FUNCTION_BLOCK FB_StatesTest
VAR_INPUT
	xboVectorTargetReached : BOOL;
	xinSatus : INT;
END_VAR
VAR_OUTPUT
	yinControl : RobotControl;
	ysTargetPosition : sPosition;
	yinTargetMap : INT;
END_VAR
VAR
	sStates : sStatesForTest;
	tonDelayWait : TON;
	tonDelayTargetReach : TON;
END_VAR
VAR CONSTANT
	//Robby 3
	creTarget1X : REAL := 628.1;
	creTarget1Y : REAL := 2668.6;
	creTarget1Phi : REAL := 0.4;
	creTarget2X : REAL := 1067.3;
	creTarget2Y : REAL := 2672.3;
	creTarget2Phi : REAL := -179.6;
	
END_VAR

CASE sStates OF
	
	sStatesForTest.Target1Vektor : 
	Gripper.closeGripperCommand := FALSE;
		yinTargetMap := 1;
		IF xboVectorTargetReached THEN 
			sStates := sStatesForTest.CoordinatesInFrontOfTarget1;
		END_IF;
		
	sStatesForTest.CoordinatesInFrontOfTarget1 :
		ysTargetPosition.reX := creTarget1X - 100;
		ysTargetPosition.reY := creTarget1Y;
		ysTargetPosition.reWinkel := creTarget1Phi;
		IF xinSatus = 3 THEN 
			sStates := sStatesForTest.Wait1;
		END_IF;
		
	sStatesForTest.Wait1 : 
	
	

		ysTargetPosition.reX := creTarget1X;
		IF 	xinSatus = 1 AND tonDelayWait.Q THEN 
			sStates := sStatesForTest.Target1;
		END_IF
		
	sStatesForTest.Target1 :
		
		IF xinSatus = 3 THEN 
			sStates := sStatesForTest.Wait2;
		END_IF;
		
	sStatesForTest.Wait2 : 
		Gripper.closeGripperCommand := TRUE;
		ysTargetPosition.reX := creTarget1X - 100;
		IF 	xinSatus = 1 AND tonDelayWait.Q THEN 
			sStates := sStatesForTest.AfterTarget1;
		END_IF
		
	sStatesForTest.AfterTarget1 :
		
		IF xinSatus = 3 THEN 
			sStates := sStatesForTest.Target2Vector;
		END_IF;
		
	sStatesForTest.Target2Vector :
	
		yinTargetMap := 2;
		IF xboVectorTargetReached THEN 
			sStates := sStatesForTest.CoordinatesInFrontOfTarget2;
		END_IF;
		
	sStatesForTest.CoordinatesInFrontOfTarget2 :
		ysTargetPosition.reX := creTarget2X + 100;
		ysTargetPosition.reY := creTarget2Y;
		ysTargetPosition.reWinkel := creTarget2Phi;
		IF xinSatus = 3 THEN 
			sStates := sStatesForTest.Wait3;
		END_IF;
		
		sStatesForTest.Wait3 : 
		ysTargetPosition.reX := creTarget2X;
		IF 	xinSatus = 1 AND tonDelayWait.Q THEN 
			sStates := sStatesForTest.Target2;
		END_IF	
		
	sStatesForTest.Target2 :
	
		
		IF xinSatus = 3 THEN 
			sStates := sStatesForTest.Wait4;
		END_IF;
		
		
		sStatesForTest.Wait4 : 
		Gripper.closeGripperCommand := FALSE;
		ysTargetPosition.reX := creTarget2X + 100;
		IF 	xinSatus = 1 AND tonDelayWait.Q THEN 
			sStates := sStatesForTest.AfterTarget2;
		END_IF	
		
	sStatesForTest.AfterTarget2 :
	
		IF xinSatus = 3 THEN 
			sStates := sStatesForTest.ParkingVector;
		END_IF;
		
	sStatesForTest.ParkingVector :
	
		yinTargetMap := 7;
		IF xboVectorTargetReached THEN 
			sStates := sStatesForTest.Finished;
		END_IF;
		
	sStatesForTest.Finished : ;
	
END_CASE

tonDelayWait(IN := (sStatesForTest.Wait1 = sStates) OR (sStatesForTest.Wait2 = sStates) OR (sStatesForTest.Wait3 = sStates) OR (sStatesForTest.Wait4 = sStates), PT := T#0.1S);

IF (sStatesForTest.Target1Vektor = sStates) OR (sStatesForTest.Target2Vector = sStates) OR (sStatesForTest.ParkingVector = sStates) THEN
	yinControl := 3;
END_IF

IF (sStatesForTest.CoordinatesInFrontOfTarget1 = sStates) OR (sStatesForTest.Target1 = sStates) OR (sStatesForTest.AfterTarget1 = sStates)
 OR (sStatesForTest.CoordinatesInFrontOfTarget2 = sStates) OR (sStatesForTest.Target2 = sStates) OR (sStatesForTest.AfterTarget2 = sStates) THEN
	yinControl := 4;
END_IF

IF (sStatesForTest.Finished = sStates) THEN
	yinControl := 1;
END_IF

IF (sStatesForTest.Wait1 = sStates) OR (sStatesForTest.Wait2 = sStates) OR (sStatesForTest.Wait3 = sStates) OR (sStatesForTest.Wait4 = sStates) THEN
	yinControl := 0;
END_IF

END_FUNCTION_BLOCK

(* stored: Version 1.1.0.1, ProductVersion 3.1.4026.13
   POU FB_StatesTest: Id {df968e2c-77cc-4fca-870b-fcefcbefbe3f}, SpecialFunc None *)
